// TIA Portal V19 export
TYPE "ValveAlr"
// stored: Access Published
   STRUCT
      TimeOutRest : Bool;   // Time out of rest command
      TimeOutWork : Bool;   // Time out of work command
      LimitSwitches : Bool;   // Both limit switch togheter on
   END_STRUCT;
END_TYPE
